# B&R Automation Studio project rebelS1
Automation Studio 4.5.2.102

## Configuration Config_rebelS

CPU X20CP1382-RT, AutomationRuntime D4.52, Build 4.1.2, Vc V4.52.0

### Task classes (Cpu.sw)
```
Cyclic#4:
  Sensor_rea <- Sensor_reading.prg
  Stand_cont <- Stand_control.prg
  Communicat <- Communication.prg
Libraries: AsUDP, runtime, ComauLib, asstring
```

### Hardware
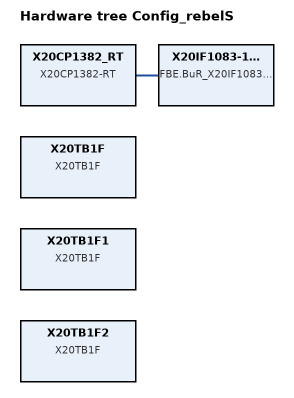
```
X20CP1382_RT : X20CP1382-RT v1.6.2.0  [X1 -> X1.SL; X2 -> X2.SL; X3 -> X3.SL]
  Module X1 (Type=X1, Virtual=true, Version=1.6.2.0)
    Connection (Connector=SS1, TargetModule=X20TB1F, TargetConnector=SS)
    Connection (Connector=SL, TargetModule=X20CP1382_RT, TargetConnector=X1)
    X1AI_ChannelType01 = 4 to 20mA
    X1AI_ChannelType02 = 4 to 20mA
  Module X2 (Type=X2, Virtual=true, Version=1.6.2.0)
    Connection (Connector=SS1, TargetModule=X20TB1F1, TargetConnector=SS)
    Connection (Connector=SL, TargetModule=X20CP1382_RT, TargetConnector=X2)
  Module X3 (Type=X3, Virtual=true, Version=1.6.2.0)
    Connection (Connector=SS1, TargetModule=X20TB1F2, TargetConnector=SS)
    Connection (Connector=SL, TargetModule=X20CP1382_RT, TargetConnector=X3)
  Connector IF2:
    ActivateDevice = 1
    Mode = Manual
    InternetAddress = 11.1.48.51
    SubnetMask = 255.255.255.0
    InaNodeNumber = 1
  Connector IF3:
    EplNatSubnet = 192.168.100.0
  ConfigurationID = rebelS_Config_rebelS
  ReActionTaskDisabled = FALSE
X20IF1083-1_COMAU_64 : FBE.BuR_X20IF1083_1_COMAU_64_the_right_ver v1.0 (OrderNumber=X20IF1083-1_COMAU_64)  [PLK1 -> X20CP1382_RT.IF3 (NodeNumber=146) [Cable Type=PowerlinkCable, Length=10, Version=1.0.0.2]]
  Supervision = off
X20TB1F : X20TB1F v1.0.0.0
X20TB1F1 : X20TB1F v1.0.0.0
X20TB1F2 : X20TB1F v1.0.0.0
```

### IoMap.iom - X20CP1382_RT/IoMap.iom
```iecst
VAR_CONFIG
	::XUAH0203S_status AT %IX."X2".DigitalInput13;
	::XUK8TAE2MM12_value AT %IW."X1".AnalogInput01;
	::XX930A2A2M12_value AT %IW."X1".AnalogInput02;
	::XS7D1A1PAL2_status AT %IX."X2".DigitalInput05;
	::XT118B1PCL2_status AT %IX."X1".DigitalInput04;
	::ODGA44A5_status AT %IX."X1".DigitalInput01;
	::XUB9BPANL2_status AT %IX."X2".DigitalInput11;
	::Robot.EPLInterface.DO1_l2014ln  AT %IB."X20IF1083-1_COMAU_64".DO1_I2014In;
	::Robot.EPLInterface.OutRealY_l2016ln  AT %ID."X20IF1083-1_COMAU_64".OutRealY_I2016In;
	::Robot.EPLInterface.OutRealX_l2015ln  AT %ID."X20IF1083-1_COMAU_64".OutRealX_I2015In;
	::Robot.EPLInterface.OutRealZ_l2017ln  AT %ID."X20IF1083-1_COMAU_64".OutRealZ_I2017In;
	 ::Robot.EPLInterface.OutRealA_l2018ln AT %ID."X20IF1083-1_COMAU_64".OutRealA_I2018In;
	::Robot.EPLInterface.OutRealE_l2019ln  AT %ID."X20IF1083-1_COMAU_64".OutRealE_I2019In;
	::Robot.EPLInterface.OutRealR_l201Aln  AT %ID."X20IF1083-1_COMAU_64".OutRealR_I201AIn;
	::Robot.EPLInterface.OutJoint1Real_l201Bln  AT %ID."X20IF1083-1_COMAU_64".OutJoint1Real_I201BIn;
	::Robot.EPLInterface.OutJoint2Real_l201Cln  AT %ID."X20IF1083-1_COMAU_64".OutJoint2Real_I201CIn;
	::Robot.EPLInterface.OutJoint3Real_l201Dln  AT %ID."X20IF1083-1_COMAU_64".OutJoint3Real_I201DIn;
	::Robot.EPLInterface.OutJoint4Real_l201Eln  AT %ID."X20IF1083-1_COMAU_64".OutJoint4Real_I201EIn;
	::Robot.EPLInterface.OutJoint5Real_l201Fln  AT %ID."X20IF1083-1_COMAU_64".OutJoint5Real_I201FIn;
	::Robot.EPLInterface.OutJoint6Real_l2020ln  AT %ID."X20IF1083-1_COMAU_64".OutJoint6Real_I2020In;
	::Robot.EPLInterface.OutDint1_l2022ln  AT %ID."X20IF1083-1_COMAU_64".OutDint1_I2022In;
	::Robot.EPLInterface.OutSmth_l2021ln  AT %ID."X20IF1083-1_COMAU_64".OutSmth_I2021In;
	::Robot.EPLInterface.OutDint2_l2023ln  AT %ID."X20IF1083-1_COMAU_64".OutDint2_I2023In;
	::Robot.EPLInterface.OutFlag1_l2024In  AT %IB."X20IF1083-1_COMAU_64".OutFlag1_I2024In;
	::Robot.EPLInterface.OutFlag2_l2025In  AT %IB."X20IF1083-1_COMAU_64".OutFlag2_I2025In;
	::Robot.EPLInterface.DO2_l2026ln  AT %IB."X20IF1083-1_COMAU_64".DO2_I2026In;
	::Robot.EPLInterface.DI1_I2001Out  AT %QB."X20IF1083-1_COMAU_64".DI1_I2001Out;
	::Robot.EPLInterface.InMotionTypeINT_l2002Out  AT %QD."X20IF1083-1_COMAU_64".InMotionTypeINT_I2002Out;
	::Robot.EPLInterface.InDintPaleteID_l2003Out  AT %QD."X20IF1083-1_COMAU_64".InDintPaleteID_I2003Out;
	::Robot.EPLInterface.InDintX_l2004Out  AT %QD."X20IF1083-1_COMAU_64".InDintX_I2004Out;
	::Robot.EPLInterface.InDintY_l2005Out  AT %QD."X20IF1083-1_COMAU_64".InDintY_I2005Out;
	::Robot.EPLInterface.InDintZ_l2006Out  AT %QD."X20IF1083-1_COMAU_64".InDintZ_I2006Out;
	::Robot.EPLInterface.InDintA_l2007Out  AT %QD."X20IF1083-1_COMAU_64".InDintA_I2007Out;
	::Robot.EPLInterface.InDintE_l2008Out  AT %QD."X20IF1083-1_COMAU_64".InDintE_I2008Out;
	::Robot.EPLInterface.InDintR_l2009Out  AT %QD."X20IF1083-1_COMAU_64".InDintR_I2009Out;
	::Robot.EPLInterface.InDintJoint1_l200AOut  AT %QD."X20IF1083-1_COMAU_64".InDintJoint1_I200AOut;
	::Robot.EPLInterface.InDintJoint2_l200BOut  AT %QD."X20IF1083-1_COMAU_64".InDintJoint2_I200BOut;
	::Robot.EPLInterface.InDintJoint3_l200COut  AT %QD."X20IF1083-1_COMAU_64".InDintJoint3_I200COut;
	::Robot.EPLInterface.InDintJoint4_l200DOut  AT %QD."X20IF1083-1_COMAU_64".InDintJoint4_I200DOut;
	::Robot.EPLInterface.InDintJoint5_l200EOut  AT %QD."X20IF1083-1_COMAU_64".InDintJoint5_I200EOut;
	::Robot.EPLInterface.InDintJoint6_l200FOut  AT %QD."X20IF1083-1_COMAU_64".InDintJoint6_I200FOut;
	::Robot.EPLInterface.InDintSmth_l2010Out  AT %QD."X20IF1083-1_COMAU_64".InDintSmth_I2010Out;
	::Robot.EPLInterface.InFlag1_l2011Out  AT %QB."X20IF1083-1_COMAU_64".InFlag1_I2011Out;
	::Robot.EPLInterface.InFlag2_l2012Out  AT %QB."X20IF1083-1_COMAU_64".InFlag2_I2012Out;
	::Robot.EPLInterface.DI2_I2013Out  AT %QB."X20IF1083-1_COMAU_64".DI2_I2013Out;
END_VAR
```

## Logical view

Binary libraries used (declarations not repeated): operator, runtime, astime, AsIecCon, AsUDP, asstring

### Global.var - Global variables
```iecst
VAR
	Robot : FBComauRobot;
	xcoord : REAL;
	palNum : INT;
	typeOfFunctionality : USINT;
	XX930A2A2M12_value : INT; (*The analog value from ultrasonic distance meter*)
	XUK8TAE2MM12_value : INT; (*The analog value from laser distance meter*)
	XUAH0203S_status : BOOL; (*The discrete output of photosensor's emitter*)
	XS7D1A1PAL2_status : BOOL; (*The discrete output of Inductive sensor*)
	ODGA44A5_status : BOOL; (*The discrete output of contrast tag's sensor*)
	XT118B1PCL2_status : BOOL; (*The discrete output of capacitive sensor*)
	XUB9BPANL2_status : BOOL; (*The discrete output of Photo-electric sensor*)
	ultrasonicDistance : REAL;
	laserDistance : REAL;
END_VAR
VAR CONSTANT
	laserCoef : REAL := 8965.486725663;
	ultrasonicCoef : REAL := 17195.1871657754;
END_VAR
VAR
	outputBeginPackFlag : BOOL;
	motionType : DINT;
	targetCoordX : INT;
	targetCoordY : INT;
	targetCoordZ : REAL;
	targetCoordA : REAL;
	targetCoordE : REAL;
	targetCoordR : REAL;
	targetAngleJ1 : REAL;
	targetAngleJ2 : REAL;
	targetAngleJ3 : REAL;
	targetAngleJ4 : REAL;
	targetAngleJ5 : REAL;
	targetAngleJ6 : REAL;
	outputEndPackFlag : BOOL;
END_VAR
```

### Package Logical/Libraries - Global libraries

### Library Logical/Libraries/ComauLib (ANSIC)

#### Types.typ - Exported data types
```iecst
TYPE
	TComauControl : 	STRUCT
		Target : TComauTarget;
		Move : BOOL;
		Homing : BOOL;
	END_STRUCT;
	TComauRobotEPLInterface : 	STRUCT
		DI1_I2001Out : USINT;
		InMotionTypeINT_l2002Out : DINT; (*2 - demo motion, 254 - ultrasonic distance sensor, 253 - laser distance sensor, 252 - *)
		InDintPaleteID_l2003Out : DINT;
		InDintX_l2004Out : DINT;
		InDintY_l2005Out : DINT;
		InDintZ_l2006Out : DINT;
		InDintA_l2007Out : DINT;
		InDintE_l2008Out : DINT;
		InDintR_l2009Out : DINT;
		InDintJoint1_l200AOut : DINT;
		InDintJoint2_l200BOut : DINT;
		InDintJoint3_l200COut : DINT;
		InDintJoint4_l200DOut : DINT;
		InDintJoint5_l200EOut : DINT;
		InDintJoint6_l200FOut : DINT;
		InDintSmth_l2010Out : DINT;
		InFlag1_l2011Out : USINT;
		InFlag2_l2012Out : USINT;
		DI2_I2013Out : USINT;
		DO1_l2014ln : USINT;
		OutRealX_l2015ln : DINT;
		OutRealY_l2016ln : DINT;
		OutRealZ_l2017ln : DINT;
		OutRealA_l2018ln : DINT;
		OutRealE_l2019ln : DINT;
		OutRealR_l201Aln : DINT;
		OutJoint1Real_l201Bln : DINT;
		OutJoint2Real_l201Cln : DINT;
		OutJoint3Real_l201Dln : DINT;
		OutJoint4Real_l201Eln : DINT;
		OutJoint5Real_l201Fln : DINT;
		OutJoint6Real_l2020ln : DINT;
		OutSmth_l2021ln : DINT;
		OutDint1_l2022ln : DINT;
		OutDint2_l2023ln : DINT;
		OutFlag1_l2024In : USINT;
		OutFlag2_l2025In : USINT;
		DO2_l2026ln : USINT;
	END_STRUCT;
	TComauRobotState :
		(
		ST_CR_IDLE,
		ST_CR_MOVE,
		Init,
		ST_CR_TAKING,
		ST_CR_RETURN
		);
	TComauTarget : 	STRUCT
		x : REAL;
		y : REAL;
		z : REAL;
		a : REAL;
		e : REAL;
		r : REAL;
		j1 : REAL;
		j2 : REAL;
		j3 : REAL;
		j4 : REAL;
		j5 : REAL;
		j6 : REAL;
	END_STRUCT;
END_TYPE
```

#### ComauLib.fun - Exported functions and function blocks
```iecst
{REDUND_ERROR} FUNCTION_BLOCK FBComauRobot (*ComauRobot function block*) (*$GROUP=User,$CAT=User,$GROUPICON=User.png,$CATICON=User.png*)
	VAR_INPUT
		Init : {REDUND_UNREPLICABLE} BOOL;
	END_VAR
	VAR_OUTPUT
		State : TComauRobotState := 1;
		EPLInterface : TComauRobotEPLInterface;
	END_VAR
	VAR_INPUT
		Control : TComauControl;
	END_VAR
END_FUNCTION_BLOCK
```

#### FBComauRobot.c
```c
#include <bur/plctypes.h>
#ifdef __cplusplus
	extern "C"
	{
#endif
	#include "ComauLib.h"
#ifdef __cplusplus
	};
#endif
/* ComauRobot function block */
void FBComauRobot(struct FBComauRobot* inst)
{
	if(inst->Init)
	{
		inst->EPLInterface.DI1_I2001Out=0;
		inst->EPLInterface.InMotionTypeINT_l2002Out = 0;
		inst->EPLInterface.InDintPaleteID_l2003Out = 0;

		inst->EPLInterface.InDintX_l2004Out = 317 * 1000;
		inst->EPLInterface.InDintY_l2005Out = 279 * 1000;
		inst->EPLInterface.InDintZ_l2006Out = 44 * 1000;
		inst->EPLInterface.InDintA_l2007Out = -81.625 * 1000;
		inst->EPLInterface.InDintE_l2008Out = 100.529 * 1000;
		inst->EPLInterface.InDintR_l2009Out = 92.591 * 1000;

		inst->EPLInterface.InDintJoint1_l200AOut = -0.063 * 1000;
		inst->EPLInterface.InDintJoint2_l200BOut = -0.541 * 1000;
		inst->EPLInterface.InDintJoint3_l200COut = -90.429 * 1000;
		inst->EPLInterface.InDintJoint4_l200DOut = -0.213 * 1000;
		inst->EPLInterface.InDintJoint5_l200EOut = -86.496 * 1000;
		inst->EPLInterface.InDintJoint6_l200FOut = -1.971 * 1000;

		inst->Init=0;
		inst->State=ST_CR_IDLE;
		return;
	}

	switch (inst->State)
	{
		/*case ST_CR_HOMING:
			inst->EPLInterface.DI1_I2001Out=1;
			inst->EPLInterface.InDintX_l2004Out = 317 * 1000;
			inst->EPLInterface.InDintY_l2005Out = 279 * 1000;
			inst->EPLInterface.InDintZ_l2006Out = 44 * 1000;
			inst->EPLInterface.InDintA_l2007Out = -81 * 1000;
			inst->EPLInterface.InDintE_l2008Out = 100 * 1000;
			inst->EPLInterface.InDintR_l2009Out = 92.591 * 1000;
			inst->Control.Move=0;
			inst->State=ST_CR_IDLE;
			break;*/
		case ST_CR_MOVE:
			if(inst->EPLInterface.DO2_l2026ln == 0)
			{
				inst->EPLInterface.DI1_I2001Out = 0;
				inst->State=ST_CR_IDLE;
			}

			break;
		case ST_CR_IDLE:
			if(inst->Control.Move == 1 && inst->EPLInterface.DO2_l2026ln == 1	)
			{
				inst->EPLInterface.DI1_I2001Out=1;
				inst->EPLInterface.InDintX_l2004Out = inst->Control.Target.x;
				inst->EPLInterface.InDintY_l2005Out = inst->Control.Target.y;
				inst->EPLInterface.InDintZ_l2006Out = inst->Control.Target.z;
				inst->EPLInterface.InDintA_l2007Out = inst->Control.Target.a;
				inst->EPLInterface.InDintE_l2008Out = inst->Control.Target.e;
				inst->EPLInterface.InDintR_l2009Out = inst->Control.Target.r;
				inst->Control.Move=0;
				inst->State=ST_CR_MOVE;
			}
			break;
		case ST_CR_TAKING:
			if(inst->EPLInterface.DO2_l2026ln == 1 && inst->Control.Move == 1)
			{
				inst->EPLInterface.DI1_I2001Out=1;
			}
			break;
	}
}
```

### Program Logical/Sensor_reading (ANSIC)

#### Main.c
```c
#include <bur/plctypes.h>

#ifdef _DEFAULT_INCLUDES
	#include <AsDefault.h>
#endif

void _INIT ProgramInit(void)
{
	typeOfFunctionality = 0;
}

void _CYCLIC ProgramCyclic(void)
{
	laserDistance = XUK8TAE2MM12_value/laserCoef;
	ultrasonicDistance = XX930A2A2M12_value/ultrasonicCoef;

}

void _EXIT ProgramExit(void)
{

}
```

### Program Logical/Stand_control (ANSIC)

#### Variables.var
```iecst
VAR
	paleteID : USINT;
	sensorID : USINT;
	i : DINT;
END_VAR
```

#### Main.c
```c
#include <bur/plctypes.h>

#ifdef _DEFAULT_INCLUDES
	#include <AsDefault.h>
#endif

void _INIT ProgramInit(void)
{
	typeOfFunctionality = 0;
	palNum = 1;
	xcoord = 421;
	Robot.Init=1;
	FBComauRobot(&Robot);
	i = 0;
}

void _CYCLIC ProgramCyclic(void)
{
	/*
	if (typeOfFunctionality == 0)
	{
		Robot.EPLInterface.InMotionTypeINT_l2002Out = 0;
		//insert your code here
		FBComauRobot(&Robot);
	}

	else if(typeOfFunctionality == 1)
	{
		Robot.EPLInterface.InMotionTypeINT_l2002Out = 1;
		//Robot.EPLInterface.InMotionTypeINT_l2002Out = motionType;
		FBComauRobot(&Robot);

		if(Robot.State == ST_CR_IDLE && Robot.EPLInterface.DO2_l2026ln == 1)
		{
			if(palNum == 1)
			{
				xcoord = 421;
			}
			else if(palNum == 10)
			{
				palNum = 1;
				xcoord = 421;
			}
			else
			{
				xcoord = xcoord - 30;
			}
			switch(i)
			{
				case 0:
					Robot.Control.Target.x = xcoord * 1000;
					Robot.Control.Target.y = 396 * 1000;
					Robot.Control.Target.z = 130 * 1000;
					Robot.Control.Target.a = 0 * 1000;
					Robot.Control.Target.e = 180 * 1000;
					Robot.Control.Target.r = 10.814 * 1000;
					Robot.Control.Move=1;
					FBComauRobot(&Robot);
					i++;
					break;
				case 1:
					Robot.Control.Target.x = xcoord * 1000;
					Robot.Control.Target.y = 396 * 1000;
					Robot.Control.Target.z = 46 * 1000;
					Robot.Control.Target.a = 0;
					Robot.Control.Target.e = 180 * 1000;
					Robot.Control.Target.r = 10.814 * 1000;
					Robot.Control.Move=1;
					FBComauRobot(&Robot);
					i++;
					break;
				case 2:
					Robot.Control.Target.x = xcoord * 1000;
					Robot.Control.Target.y = 396 * 1000;
					Robot.Control.Target.z = 130 * 1000;
					Robot.Control.Target.a = 0;
					Robot.Control.Target.e = 100 * 1000;
					Robot.Control.Target.r = 10.814 * 1000;
					Robot.Control.Move=1;
					FBComauRobot(&Robot);
					i++;
					break;
				case 3:
					Robot.Control.Target.x = 400 * 1000;
					Robot.Control.Target.y = 214.546 * 1000;
					Robot.Control.Target.z = 102.642 * 1000;
					Robot.Control.Target.a = 0;
					Robot.Control.Target.e = 180 * 1000;
					Robot.Control.Target.r = 10.814 * 1000;
					Robot.Control.Move=1;
					FBComauRobot(&Robot);
					i++;
					break;
				case 4:
					Robot.Control.Target.x = 710 * 1000;
					Robot.Control.Target.y = 214.546 * 1000;
					Robot.Control.Target.z = 102.642 * 1000;
					Robot.Control.Target.a = 0;
					Robot.Control.Target.e = 180 * 1000;
					Robot.Control.Target.r = 10.814 * 1000;
					Robot.Control.Move=1;
					FBComauRobot(&Robot);
					i++;
					break;
				case 5:
					Robot.Control.Target.x = 710 * 1000;
					Robot.Control.Target.y = -195.093 * 1000;
					Robot.Control.Target.z = 102.642 * 1000;
					Robot.Control.Target.a = 0;
					Robot.Control.Target.e = 180 * 1000;
					Robot.Control.Target.r = 10.814 * 1000;
					Robot.Control.Move=1;
					FBComauRobot(&Robot);
					i = 0;
					break;
				/*dfsadsadsadsadsadsad*/
		/*		case 6:
					Robot.Control.Target.x = 501 * 1000;
					Robot.Control.Target.y = -195.093 * 1000;
					Robot.Control.Target.z = 102.642 * 1000;
					Robot.Control.Target.a = 0;
					Robot.Control.Target.e = 180 * 1000;
					Robot.Control.Target.r = 10.814 * 1000;
					Robot.Control.Move=1;
					FBComauRobot(&Robot);
					i = 0;
					break;
				case 7:
					Robot.Control.Target.x = 501 * 1000;
					Robot.Control.Target.y = -195.093 * 1000;
					Robot.Control.Target.z = 60 * 1000;
					Robot.Control.Target.a = 0;
					Robot.Control.Target.e = 180 * 1000;
					Robot.Control.Target.r = 100.814 * 1000;
					Robot.Control.Move=1;
					FBComauRobot(&Robot);
					i = 0;
					break;
				case 8:
					Robot.Control.Target.x = 501 * 1000;
					Robot.Control.Target.y = -450 * 1000;
					Robot.Control.Target.z = 60 * 1000;
					Robot.Control.Target.a = 0;
					Robot.Control.Target.e = 180 * 1000;
					Robot.Control.Target.r = 100.814 * 1000;
					Robot.Control.Move=1;
					FBComauRobot(&Robot);
					i = 0;
					break;
				case 9:
					Robot.Control.Target.x = 501 * 1000;
					Robot.Control.Target.y = 0;
					Robot.Control.Target.z = 60 * 1000;
					Robot.Control.Target.a = 0;
					Robot.Control.Target.e = 180 * 1000;
					Robot.Control.Target.r = 100.814 * 1000;
					Robot.Control.Move=1;
					FBComauRobot(&Robot);
					i = 0;
					break;
				case 10:
					Robot.Control.Target.x = 341 * 1000;
					Robot.Control.Target.y = 0;
					Robot.Control.Target.z = 60 * 1000;
					Robot.Control.Target.a = 0;
					Robot.Control.Target.e = 180 * 1000;
					Robot.Control.Target.r = 100.814 * 1000;
					Robot.Control.Move=1;
					FBComauRobot(&Robot);
					i = 0;
					break;
				/* sadsadwdddwsferf */
		/*		case 11:
					Robot.Control.Target.x = 341 * 1000;
					Robot.Control.Target.y = -450 * 1000;
					Robot.Control.Target.z = 60 * 1000;
					Robot.Control.Target.a = 0;
					Robot.Control.Target.e = 180 * 1000;
					Robot.Control.Target.r = 100.814 * 1000;
					Robot.Control.Move=1;
					FBComauRobot(&Robot);
					i = 0;
					break;
				case 12:
					Robot.Control.Target.x = 181 * 1000;
					Robot.Control.Target.y = -450 * 1000;
					Robot.Control.Target.z = 60 * 1000;
					Robot.Control.Target.a = 0;
					Robot.Control.Target.e = 180 * 1000;
					Robot.Control.Target.r = 100.814 * 1000;
					Robot.Control.Move=1;
					FBComauRobot(&Robot);
					i = 0;
					break;
				case 13:
					Robot.Control.Target.x = 181 * 1000;
					Robot.Control.Target.y = -210;
					Robot.Control.Target.z = 60 * 1000;
					Robot.Control.Target.a = 0;
					Robot.Control.Target.e = 180 * 1000;
					Robot.Control.Target.r = 100.814 * 1000;
					Robot.Control.Move=1;
					FBComauRobot(&Robot);
					i = 0;
					break;

				case 14:
					Robot.Control.Target.x = 501 * 1000;
					Robot.Control.Target.y = -205;
					Robot.Control.Target.z = 60 * 1000;
					Robot.Control.Target.a = 0;
					Robot.Control.Target.e = 180 * 1000;
					Robot.Control.Target.r = 10.814 * 1000;
					Robot.Control.Move=1;
					FBComauRobot(&Robot);
					i = 0;
					break;

				case 15:
					Robot.Control.Target.x = xcoord * 1000;
					Robot.Control.Target.y = 396 * 1000;
					Robot.Control.Target.z = 130 * 1000;
					Robot.Control.Target.a = 0;
					Robot.Control.Target.e = 180 * 1000;
					Robot.Control.Target.r = 10.814 * 1000;
					Robot.Control.Move=1;
					FBComauRobot(&Robot);
					i = 0;
					break;

				case 16:
					Robot.Control.Target.x = xcoord * 1000;
					Robot.Control.Target.y = 396 * 1000;
					Robot.Control.Target.z = 46 * 1000;
					Robot.Control.Target.a = 0;
					Robot.Control.Target.e = 180 * 1000;
					Robot.Control.Target.r = 10.814 * 1000;
					Robot.Control.Move=1;
					FBComauRobot(&Robot);
					i = 0;
					break;

				case 17:
					Robot.Control.Target.x = xcoord * 1000;
					Robot.Control.Target.y = 396 * 1000;
					Robot.Control.Target.z = 130 * 1000;
					Robot.Control.Target.a = 0;
					Robot.Control.Target.e = 180 * 1000;
					Robot.Control.Target.r = 10.814 * 1000;
					Robot.Control.Move=1;
					FBComauRobot(&Robot);
					i = 0;
					break;
					palNum++;
			}
		}

		else if (typeOfFunctionality == 2)
		{
			Robot.EPLInterface.InMotionTypeINT_l2002Out = 0;
			//insert your code here
			FBComauRobot(&Robot);
		}
		else if (typeOfFunctionality == 3)
		{
			Robot.EPLInterface.InMotionTypeINT_l2002Out = 0;
			//insert your code here
			FBComauRobot(&Robot);
		}
	}*/
}

void _EXIT ProgramExit(void)
{

}

void examineSensor(senID, palID)
{

}
```

### Program Logical/Communication (ANSIC)

#### Types.typ
```iecst
TYPE
	Server_typ : 	STRUCT  (*UDP Server Variables*)
		sStep : UINT; (*UDP Server Step Variable*)
		client_address : STRING[20]; (*Address of the client connection to the Server*)
		UdpOpen_1 : UdpOpen; (*AsUDP.UdpOpen FUB*)
		UdpConnect_1 : UdpConnect; (*AsUDP.UdpConnect FUB*)
		UdpSend_1 : UdpSend; (*AsUDP.UdpSend FUB*)
		UdpRecv_1 : UdpRecv; (*AsUDP.UdpRecv FUB*)
		UdpDisconnect_1 : UdpDisconnect; (*AsUDP.UdpDisconnect FUB*)
		UdpClose_1 : UdpClose; (*AsUDP.UdpClose FUB*)
		outData_buffer : ARRAY[0..100]OF UDINT; (*Data buffer ( receive and send )*)
		privClient : STRING[20];
		inData_buffer : ARRAY[0..100]OF UDINT;
	END_STRUCT;
END_TYPE
```

#### Variables.var
```iecst
VAR
	cutBuf : STRING[7];
	Server_1 : Server_typ;
	buff : STRING[6];
	p : STRING[1];
	intRobX : INT;
	intRobY : INT;
	intRobZ : INT;
	intRobA : INT;
	intRobE : INT;
	intRobR : INT;
	intRobJ1 : INT;
	intRobJ2 : INT;
	intRobJ3 : INT;
	intRobJ4 : INT;
	intRobJ5 : INT;
	intRobJ6 : INT;
	outIntValue1 : INT;
	outIntValue2 : INT;
	outIntValue3 : INT;
	outIntFlag1 : INT;
	outIntFlag2 : INT;
	outIntEndPackFlag : INT;
END_VAR
```

#### Main.c
```c
#include <bur/plctypes.h>

#ifdef _DEFAULT_INCLUDES
	#include <AsDefault.h>
#endif

void packData()
{
	memset(Server_1.outData_buffer, 0, sizeof(Server_1.outData_buffer));

	strcat (Server_1.outData_buffer, "sensors: ");

	itoa(laserDistance, &buff);
	strcat (Server_1.outData_buffer, buff);
	strcat (Server_1.outData_buffer, ", ");

	itoa(ultrasonicDistance, &buff);
	strcat (Server_1.outData_buffer, buff);
	strcat (Server_1.outData_buffer, ", ");

	itoa(XUAH0203S_status, &buff); //photosensor
	strcat (Server_1.outData_buffer, buff);
	strcat (Server_1.outData_buffer, ", ");

	itoa(XS7D1A1PAL2_status, &buff); //inductive sensor
	strcat (Server_1.outData_buffer, buff);
	strcat (Server_1.outData_buffer, ", ");

	itoa(ODGA44A5_status, &buff); //contrast tag sensor
	strcat (Server_1.outData_buffer, buff);
	strcat (Server_1.outData_buffer, ", ");

	itoa(XT118B1PCL2_status, &buff); //capacitive sensor
	strcat (Server_1.outData_buffer, buff);
	strcat (Server_1.outData_buffer, ", ");

	itoa(XUB9BPANL2_status, &buff); //photoelectric sensor
	strcat (Server_1.outData_buffer, buff);

	//the end of data pack
	strcat (Server_1.outData_buffer, ";");
}

void _INIT ProgramInit(void)
{

}

void _CYCLIC ProgramCyclic(void)
{
	switch(Server_1.sStep)
	{
		case 0:
			Server_1.UdpOpen_1.enable = 1;
			Server_1.UdpOpen_1.pIfAddr = 0;
			Server_1.UdpOpen_1.port = 12051;
			Server_1.UdpOpen_1.options = 0;
			UdpOpen(&Server_1.UdpOpen_1);

			if(Server_1.UdpOpen_1.status == 0)
			{
				Server_1.sStep = 1;
			}
			else if (Server_1.UdpOpen_1.status == ERR_FUB_BUSY)
			{

			}
			else  //(* Goto Error Step *)
			{
				Server_1.sStep = 10;
			}
			break;
		case 1:
			Server_1.UdpRecv_1.enable = 1;
			Server_1.UdpRecv_1.ident = Server_1.UdpOpen_1.ident;	//(* Client Ident from AsUDP.UDP_Open *)
			Server_1.UdpRecv_1.pData = (UDINT)&Server_1.inData_buffer[0];	//(* Where to store the incoming data *)
			Server_1.UdpRecv_1.datamax = sizeof(Server_1.inData_buffer);	//(* Lenght of data buffer *)
			Server_1.UdpRecv_1.flags = 0;
			Server_1.UdpRecv_1.pIpAddr = (UDINT)&Server_1.client_address[0];	//(* IP Address of the Client *)
			UdpRecv(&Server_1.UdpRecv_1);	//(* Call the Function*)

			if(Server_1.UdpRecv_1.status == 0)  //(* Data received *)
			{
				Server_1.sStep = 2;
			}
			else if (Server_1.UdpRecv_1.status == udpERR_NO_DATA)//(* No data received - wait *)
			{
				Server_1.sStep = 2;				//(* No Data received *)
			}
			else if (Server_1.UdpRecv_1.status == ERR_FUB_BUSY) //(* UdpRecv not finished -> redo *)
			{
				//(* Busy *)
			}
			else
			{
				Server_1.sStep = 10;
			}
			break;

		case 2:	//(* Send Data back to Client *)
			packData();

			Server_1.UdpSend_1.enable = 1;
			Server_1.UdpSend_1.ident = Server_1.UdpOpen_1.ident;	//(* Client Ident from AsUDP.UDP_Open *)
			Server_1.UdpSend_1.pHost = (UDINT)&Server_1.client_address[0];	//(* IP Address of the Client *)
			Server_1.UdpSend_1.port = Server_1.UdpRecv_1.port;		//(* Port number of the Client *)
			Server_1.UdpSend_1.pData = (UDINT)&Server_1.outData_buffer[0];	//(* Which data to send *)
			Server_1.UdpSend_1.datalen = sizeof(Server_1.outData_buffer);	//(* Length of data to send *)
			Server_1.UdpSend_1.flags = 0;
			UdpSend(&Server_1.UdpSend_1);	//(* Call the Function*)

			if (Server_1.UdpSend_1.status == 0)  //(* Data sent *)
			{
				Server_1.sStep = 1;
			}
			else if(Server_1.UdpSend_1.status == ERR_FUB_BUSY)  //(* UdpSend not finished -> redo *)
			{
				//(* Busy *)
			}
			else  //(* Goto Error Step *)
			{
				Server_1.sStep = 10;
			}
			break;
		case 3: //recieve data from client with checking previlige status

			break;
		case 10:
			/*TODO: ?????????? ??????*/
			break;
	}
}

void _EXIT ProgramExit(void)
{

}
```

Listed in the project but not available here: Logical/Global.typ, Logical/Libraries/ComauLib/Constants.var
